TYPE TRAJECTORY :
STRUCT
		size     	  :UINT:=0;                          //轨迹点的数目
		//points        :ARRAY[0..100] OF this_point;      //要执行的一系列轨迹点  
END_STRUCT
END_TYPE

(* stored: Version 1.1.0.1, ProductVersion 3.1.4022.10
   DUT TRAJECTORY: Id {bdbaa5f1-508e-4a9c-8490-0e519f8090a5} *)
